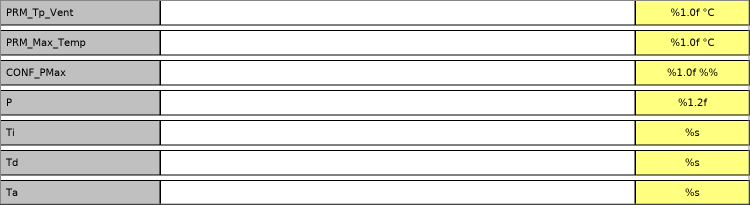
VISUALIZATION VISU_CONFIG_CHAUFF  // 750x205
(*visualistion pour secondaire dans chambre et primaire dans sas ==> paramètres pour chambre*)
VAR_IN_OUT
	m_Input_PRG_CHAUFFAGE : BLOCK_PRG_CHAUFFAGE;
END_VAR
    Rectangle (160,0 475x25), text list: 'TextList_Config_Chauffage', text index: 1
    Rectangle (635,0 115x25), "%1.0f °C", text variable: m_Input_PRG_CHAUFFAGE.PRM_Tp_Vent, input disabled if: NOT Global_Variables.PRG_USER.ACTU_USER.CONF_MACHINE
        OnMouseClick: write the text variable via VisuDialogs.Numpad, min m_Input_PRG_CHAUFFAGE.CONF_Min_Temp, max 55
    Rectangle (0,0 160x25), "PRM_Tp_Vent"
    Rectangle (160,30 475x25), text list: 'TextList_Config_Chauffage', text index: 2
    Rectangle (635,30 115x25), "%1.0f °C", text variable: m_Input_PRG_CHAUFFAGE.PRM_Max_Temp, input disabled if: NOT Global_Variables.PRG_USER.ACTU_USER.CONF_MACHINE
        OnMouseClick: write the text variable via VisuDialogs.Numpad, min m_Input_PRG_CHAUFFAGE.CONF_Min_Temp, max m_Input_PRG_CHAUFFAGE.CONF_Max_Temp
    Rectangle (0,30 160x25), "PRM_Max_Temp"
    Rectangle (160,60 475x25), text list: 'TextList_Config_Chauffage', text index: 3
    Rectangle (160,90 475x25), text list: 'TextList_Config_Chauffage', text index: 4
    Rectangle (635,60 115x25), "%1.0f %%", text variable: m_Input_PRG_CHAUFFAGE.CHAUFFAGE.CH.CONF_PMAX, input disabled if: NOT Global_Variables.PRG_USER.ACTU_USER.CONF_MACHINE
        OnMouseClick: write the text variable via VisuDialogs.Numpad, min 0, max m_Input_PRG_CHAUFFAGE.CONF_Pmax_max
    Rectangle (0,60 160x25), "CONF_PMax"
    Rectangle (635,90 115x25), "%1.2f", text variable: m_Input_PRG_CHAUFFAGE.CHAUFFAGE.CH.PRM_PID.KpHeat, input disabled if: NOT Global_Variables.PRG_USER.ACTU_USER.CONF_MACHINE
        OnMouseClick: write the text variable via VisuDialogs.Numpad, min 0
    Rectangle (0,90 160x25), "P"
    Rectangle (160,120 475x25), text list: 'TextList_Config_Chauffage', text index: 5
    Rectangle (635,120 115x25), "%s", text variable: m_Input_PRG_CHAUFFAGE.CHAUFFAGE.CH.PRM_PID.TnHeat, input disabled if: NOT Global_Variables.PRG_USER.ACTU_USER.CONF_MACHINE
        OnMouseClick: write the text variable via VisuDialogs.Keypad
    Rectangle (0,120 160x25), "Ti"
    Rectangle (0,150 160x25), "Td"
    Rectangle (160,150 475x25), text list: 'TextList_Config_Chauffage', text index: 6
    Rectangle (635,150 115x25), "%s", text variable: m_Input_PRG_CHAUFFAGE.CHAUFFAGE.CH.PRM_PID.TvHeat, input disabled if: NOT Global_Variables.PRG_USER.ACTU_USER.CONF_MACHINE
        OnMouseClick: write the text variable via VisuDialogs.Keypad
    Rectangle (0,180 160x25), "Ta"
    Rectangle (160,180 475x25), text list: 'TextList_Chauffage', text index: 6
    Rectangle (635,180 115x25), "%s", text variable: m_Input_PRG_CHAUFFAGE.CHAUFFAGE.CH.PRM_PID.TdHeat, input disabled if: NOT Global_Variables.PRG_USER.ACTU_USER.CONF_MACHINE
        OnMouseClick: write the text variable via VisuDialogs.Keypad
END_VISUALIZATION

(* stored: Version 1.1.0.1, ProductVersion 3.1.4024.10
   Visu VISU_CONFIG_CHAUFF: Id {b8d42ab6-6eb3-491a-abd1-604b2fff681a} *)
